FUNCTION_BLOCK Performance2 (* Composite Function Block Type *)
  (* Standard: 61499-2 *)
  (* Version 1.0, 2020-12-26, jetbrains *)
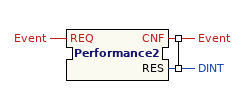
  EVENT_INPUT
    REQ; (* Normal Execution Request *)
  END_EVENT
  EVENT_OUTPUT
    CNF WITH RES; (* Execution Confirmation *)
  END_EVENT
  VAR_OUTPUT
    RES : DINT; (* Output event qualifier *)
  END_VAR
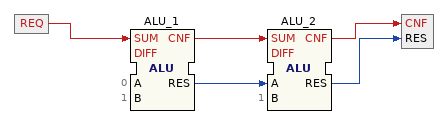
  FBS
    ALU_2 : ALU(B := 1);
    ALU_1 : ALU(A := 0, B := 1);
  END_FBS
  EVENT_CONNECTIONS
    ALU_2.CNF TO CNF;
    REQ TO ALU_1.SUM;
    ALU_1.CNF TO ALU_2.SUM;
  END_CONNECTIONS
  DATA_CONNECTIONS
    ALU_2.RES TO RES;
    ALU_1.RES TO ALU_2.A;
  END_CONNECTIONS
END_FUNCTION_BLOCK
